// TwinCAT 3 PLC project TcLog
// Title: TcLog
// Company: Benedikt Geisler
// Author: Benedikt Geisler
// ProjectVersion: 0.6.1
// Description: TcLog provides logging functionality to TwinCAT.
// ProgramVersion: 3.1.4026.20
// libraries:
//   Tc2_Standard, * (Beckhoff Automation GmbH)
//   Tc2_System, * (Beckhoff Automation GmbH)
//   Tc2_Utilities, * (Beckhoff Automation GmbH)
//   Tc3_DynamicMemory, * (Beckhoff Automation GmbH)
//   Tc3_Module, * (Beckhoff Automation GmbH)
//   TcUnit, * (www.tcunit.org)
// project tree:
//   / Constants.TcGVL
//   Logger/ LogLevelToAdsLogMsgType.TcPOU (not stored), TcLog.TcPOU, TcLogCore.TcPOU (not stored), TcLogTrig.TcPOU (not stored)
//   StringBuilder/_Interfaces/ ILimitedStringBuilder.TcIO (not stored), IStringBuilder.TcIO (not stored)
//   Utils/ AnyToString.TcPOU (not stored), DateTime.TcPOU (not stored), DeleteOldFiles.TcPOU (not stored), DynamicStringBuffer.TcPOU (not stored), GetFileAgeInSeconds.TcPOU (not stored)
//   Utils/DataTypes/ DeleteFilesState.TcDUT (not stored), PersistToFileState.TcDUT (not stored)
//   Logger/DataTypes/ ErrorCodes.TcDUT (not stored), LogLevels.TcDUT (not stored), RollingIntervals.TcDUT (not stored), Error.TcDUT (not stored), LoggingConfiguration.TcDUT (not stored)
//   Logger/Interfaces/ ILog.TcIO (not stored), ILogCore.TcIO (not stored)
//   StringBuilder/ StringBuilder.TcPOU (not stored)
// real-time tasks:
//   TASK PlcTask1: cycle T#10ms, priority 21, ADS port 351

// ---- Constants.TcGVL
{attribute 'qualified_only'}
VAR_GLOBAL CONSTANT
	/// Fifo overhead needed to manage the string buffer
	FifoOverhead : UDINT := 10;

	/// Buffer size of temporary buffer used to persist all log messages in one cycle. 
	BufferSize : UDINT := (100 * (Tc2_System.MAX_STRING_LENGTH + FifoOverhead));
END_VAR

// ---- Logger/TcLog.TcPOU
/// `TcLog` is the client side of the logger.  
///
/// It is used to send the logs to `TcLogCore`. Typically, it is instantiated
/// once in each `FUNCTION_BLOCK` or `PROGRAM` where logging is done. The same 
/// instance can then be used for all logging within that POU. 
///
/// `TcLog` implements a string builder that facilitates the compilation of the log
/// message without the need for external data type conversions or multiple chained `CONCAT` calls.
/// See the method section for more information.
///
/// The last method to call after the log message has been built is one of ´[Debug|Information|Warning|Error|Fatal]`. 
/// This sets the log level of the message and sends it off to the log message queue of `TcLogCore` where it will
/// be processed according to its configuration.
{attribute 'linkalways'}
{attribute 'hide_all_locals'}
{attribute 'reflection'} 
FUNCTION_BLOCK TcLog IMPLEMENTS ILog
VAR
  _logConditionSatisfied : BOOL; // flag that indicates, whether log condition has been satisfied.
                                // Logging will only be carried out it this evaluates to TRUE.                    
  _logDataInitialized : BOOL; // flag that indicate, whether log data has been initialized.
                             // Necessary for configuration methods to provide a fluent interface.                            
  _logData : Tc2_System.T_MaxString; // contains message to be logged.
  _usedLogger : ILogCore;
  {attribute 'instance-path'} 
  {attribute 'noinit'} 
  _instancePath : STRING; // contains instance path
END_VAR
VAR_STAT
  {attribute 'hide'}
  s_loggerSingletonInstance : ILogCore; // Wires up TcLog ("Client") to TcLogCore ("Server") (Singleton-Behaviour)
END_VAR
VAR CONSTANT
  InvalidLoggerReference : UDINT := 0;
END_VAR

/// Appends any given data to the log string. The type of the provided data
/// has to be one of the [standard data types](https://infosys.beckhoff.com/english.php?content=../content/1033/tc3_plc_intro/2529388939.html&id=).
/// This method can be chained.
METHOD AppendAny : REFERENCE TO TcLog
VAR_INPUT
  /// data to be appended to log string.
  data : ANY;
END_VAR
InitializeLogData();

_logData := Tc2_Standard.CONCAT(_logData, AnyToString(data));

AppendAny REF= THIS^;
END_METHOD

/// Appends a BYTE to the log string.
/// This method can be chained.
METHOD PUBLIC AppendByte : REFERENCE TO TcLog
VAR_INPUT
  /// data to be appended to log string.
  data : BYTE;
END_VAR
AppendByte REF= AppendString(TO_STRING(data));
END_METHOD

/// Appends a DATE to the log string.
/// This method can be chained.
METHOD PUBLIC AppendDate : REFERENCE TO TcLog
VAR_INPUT
  /// data to be appended to log string.
  data : DATE;
END_VAR
AppendDate REF= AppendString(TO_STRING(data));
END_METHOD

/// Appends a DATE_AND_TIME to the log string.
/// This method can be chained.
METHOD PUBLIC AppendDateAndTime : REFERENCE TO TcLog
VAR_INPUT
  /// data to be appended to log string.
  data : DATE_AND_TIME;
END_VAR
AppendDateAndTime REF= AppendString(TO_STRING(data));
END_METHOD

/// Appends a DINT to the log string.
/// This method can be chained.
METHOD PUBLIC AppendDint : REFERENCE TO TcLog
VAR_INPUT
  /// data to be appended to log string.
  data : DINT;
END_VAR
AppendDint REF= AppendString(TO_STRING(data));
END_METHOD

/// Appends a DWORD to the log string.
/// This method can be chained.
METHOD PUBLIC AppendDword : REFERENCE TO TcLog
VAR_INPUT
  /// data to be appended to log string.
  data : DWORD;
END_VAR
AppendDword REF= AppendString(TO_STRING(data));
END_METHOD

/// Appends an INT to the log string.
/// This method can be chained.
METHOD PUBLIC AppendInt : REFERENCE TO TcLog
VAR_INPUT
  /// data to be appended to log string.
  data : INT;
END_VAR
AppendInt REF= AppendString(TO_STRING(data));
END_METHOD

/// Appends a LDATE to the log string.
/// This method can be chained.
METHOD PUBLIC AppendLDate : REFERENCE TO TcLog
VAR_INPUT
  /// data to be appended to log string.
  data : LDATE;
END_VAR
AppendLDate REF= AppendString(TO_STRING(data));
END_METHOD

/// Appends a LDATE_AND_TIME to the log string.
/// This method can be chained.
METHOD PUBLIC AppendLDateAndTime : REFERENCE TO TcLog
VAR_INPUT
  /// data to be appended to log string.
  data : LDATE_AND_TIME;
END_VAR
AppendLDateAndTime REF= AppendString(TO_STRING(data));
END_METHOD

/// Appends an LINT to the log string.
/// This method can be chained.
METHOD PUBLIC AppendLint : REFERENCE TO TcLog
VAR_INPUT
  /// data to be appended to log string.
  data : LINT;
END_VAR
AppendLint REF= AppendString(TO_STRING(data));
END_METHOD

/// Appends an LREAL to the log string.
/// This method can be chained.
METHOD PUBLIC AppendLreal : REFERENCE TO TcLog
VAR_INPUT
  /// data to be appended to log string.
  data : LREAL;
END_VAR
AppendLreal REF= AppendString(TO_STRING(data));
END_METHOD

/// Appends a LTIME_OF_DAY to the log string.
/// This method can be chained.
METHOD PUBLIC AppendLTimeOfDay : REFERENCE TO TcLog
VAR_INPUT
  /// data to be appended to log string.
  data : LTIME_OF_DAY;
END_VAR
AppendLTimeOfDay REF= AppendString(TO_STRING(data));
END_METHOD

/// Appends an LWORD to the log string.
/// This method can be chained.
METHOD PUBLIC AppendLword : REFERENCE TO TcLog
VAR_INPUT
  /// data to be appended to log string.
  data : LWORD;
END_VAR
AppendLword REF= AppendString(TO_STRING(data));
END_METHOD

/// Appends a REAL to the log string.
/// This method can be chained.
METHOD PUBLIC AppendReal : REFERENCE TO TcLog
VAR_INPUT
  /// data to be appended to log string.
  data : REAL;
END_VAR
AppendReal REF= AppendString(TO_STRING(data));
END_METHOD

/// Appends a SINT to the log string.
/// This method can be chained.
METHOD PUBLIC AppendSint : REFERENCE TO TcLog
VAR_INPUT
  /// data to be appended to log string.
  data : SINT;
END_VAR
AppendSint REF= AppendString(TO_STRING(data));
END_METHOD

/// Appends another string to the log message.
/// This method can be chained.
METHOD AppendString : REFERENCE TO TcLog
VAR_INPUT
  /// data to be appended to log string.
  data : Tc2_System.T_MaxString; 
END_VAR
InitializeLogData();

_logData := Tc2_Standard.CONCAT(_logData, data);
  
AppendString REF= THIS^;
END_METHOD

/// Appends a TIME_OF_DAY to the log string.
/// This method can be chained.
METHOD PUBLIC AppendTimeOfDay : REFERENCE TO TcLog
VAR_INPUT
  /// data to be appended to log string.
  data : TIME_OF_DAY;
END_VAR
AppendTimeOfDay REF= AppendString(TO_STRING(data));
END_METHOD

/// Appends a UDINT to the log string.
/// This method can be chained.
METHOD PUBLIC AppendUdint : REFERENCE TO TcLog
VAR_INPUT
  /// data to be appended to log string.
  data : UDINT;
END_VAR
AppendUdint REF= AppendString(TO_STRING(data));
END_METHOD

/// Appends a UINT to the log string.
/// This method can be chained.
METHOD PUBLIC AppendUint : REFERENCE TO TcLog
VAR_INPUT
  /// data to be appended to log string.
  data : UINT;
END_VAR
AppendUint REF= AppendString(TO_STRING(data));
END_METHOD

/// Appends a ULINT to the log string.
/// This method can be chained.
METHOD PUBLIC AppendUlint : REFERENCE TO TcLog
VAR_INPUT
  /// data to be appended to log string.
  data : ULINT;
END_VAR
AppendUlint REF= AppendString(TO_STRING(data));
END_METHOD

/// Appends a USINT to the log string.
/// This method can be chained.
METHOD PUBLIC AppendUsint : REFERENCE TO TcLog
VAR_INPUT
  /// data to be appended to log string.
  data : USINT;
END_VAR
AppendUsint REF= AppendString(TO_STRING(data));
END_METHOD

/// Appends information about the given variable to the log string. 
/// This method can be chained.
/// Example: 

/// ```st
/// VAR
///   Logger: TcLog;
///    myInt : INT := 10;
///   myVarInfo : __SYSTEM.VAR_INFO := __VARINFO(myInt);
/// END_VAR
/// Logger.AppendVariable(myVarInfo, myInt);
/// ```
///
METHOD AppendVariable : REFERENCE TO TcLog
VAR_INPUT
  /// [VAR_INFO](https://infosys.beckhoff.com/index.php?content=../content/1031/tc3_plc_intro/3527777675.html&id=) of variable to be appended to log string.
  varInfo : __SYSTEM.VAR_INFO;
  /// Value of variable to be appended to log string.
  value : ANY; 
END_VAR
VAR
  format : Tc2_Utilities.FB_FormatString;
  symbolName : Tc2_System.T_MaxString;
  typeName : Tc2_System.T_MaxString;
END_VAR
InitializeLogData();

symbolName := varInfo.Symbol;
typeName := varInfo.TypeName; 

format(
  sFormat := '%s [%s] : ',
  arg1 := Tc2_Utilities.F_String(symbolName),
  arg2 := Tc2_Utilities.F_String(typeName));
  
AppendString(format.sOut);
AppendAny(value);

AppendVariable REF= THIS^;
END_METHOD

/// Appends a WORD to the log string.
/// This method can be chained.
METHOD PUBLIC AppendWord : REFERENCE TO TcLog
VAR_INPUT
  /// data to be appended to log string.
  data : WORD;
END_VAR
AppendWord REF= AppendString(TO_STRING(data));
END_METHOD

/// Logs the log string in DEBUG level.
METHOD Debug : BOOL
VAR_INPUT
  /// Message to be appended to log string.
  message : Tc2_System.T_MaxString; 
END_VAR
InitializeLogData();
IF _logConditionSatisfied THEN
  IF _usedLogger <> InvalidLoggerReference THEN 
    _usedLogger.LogStandardFormat(Tc2_Standard.CONCAT(_logData, message), ShortenInstancePath(_instancePath), LogLevels.Debug); 
  ELSE
    Tc2_System.ADSLOGSTR(ADSLOG_MSGTYPE_LOG OR LogLevelToAdsLogMsgType(LogLevels.Error), 'usedLogger: No valid reference', ''); 
  END_IF
END_IF
_logDataInitialized := FALSE;
END_METHOD

/// Logs the log string in ERROR level.
METHOD Error : BOOL
VAR_INPUT
  /// Message to be appended to log string.
  message : Tc2_System.T_MaxString; 
END_VAR
InitializeLogData();
IF _logConditionSatisfied THEN
  IF _usedLogger <> InvalidLoggerReference THEN 
    _usedLogger.LogStandardFormat(Tc2_Standard.CONCAT(_logData, message), ShortenInstancePath(_instancePath), LogLevels.Error); 
  ELSE
    Tc2_System.ADSLOGSTR(ADSLOG_MSGTYPE_LOG OR LogLevelToAdsLogMsgType(LogLevels.Error), 'usedLogger: No valid reference', ''); 
  END_IF
END_IF
_logDataInitialized := FALSE;
END_METHOD

/// Logs the log string in FATAL level.
METHOD Fatal : BOOL
VAR_INPUT
  /// Message to be appended to log string.
  message : Tc2_System.T_MaxString; 
END_VAR
InitializeLogData();
IF _logConditionSatisfied THEN
  IF _usedLogger <> InvalidLoggerReference THEN 
    _usedLogger.LogStandardFormat(Tc2_Standard.CONCAT(_logData, message), ShortenInstancePath(_instancePath), LogLevels.Fatal); 
  ELSE
    Tc2_System.ADSLOGSTR(ADSLOG_MSGTYPE_LOG OR LogLevelToAdsLogMsgType(LogLevels.Error), 'usedLogger: No valid reference', ''); 
  END_IF
END_IF
_logDataInitialized := FALSE;
END_METHOD

/// Logs the log string in INFORMATION level.
METHOD Information : BOOL
VAR_INPUT
  /// Message to be appended to log string.
  message : Tc2_System.T_MaxString; 
END_VAR
InitializeLogData();
IF _logConditionSatisfied THEN
  IF _usedLogger <> InvalidLoggerReference THEN 
    _usedLogger.LogStandardFormat(Tc2_Standard.CONCAT(_logData, message), ShortenInstancePath(_instancePath), LogLevels.Information); 
  ELSE
    Tc2_System.ADSLOGSTR(ADSLOG_MSGTYPE_LOG OR LogLevelToAdsLogMsgType(LogLevels.Error), 'usedLogger: No valid reference', ''); 
  END_IF
END_IF
_logDataInitialized := FALSE;
END_METHOD

/// Initializes the reference to the core logger. Should only be called once from the core logger directly.
METHOD PUBLIC Init : BOOL
VAR_INPUT
  /// Reference to TcLoggerCore instance.
  ref2Core : ILogCore; 
END_VAR
IF s_loggerSingletonInstance = 0 THEN
	s_loggerSingletonInstance := ref2Core;
END_IF
END_METHOD

// Necessary to provide a fluent interface of the function. 
// Has to be called at the begin of any method that returns a reference to THIS^
METHOD PRIVATE InitializeLogData : BOOL
IF NOT _logDataInitialized THEN
  _logConditionSatisfied := TRUE;
  _logData := '';
  _logDataInitialized := TRUE;
  IF _usedLogger = 0 THEN _usedLogger := s_loggerSingletonInstance; END_IF
END_IF
END_METHOD

/// Conditional execution of the log command. Only executes logging when Cond = TRUE.
METHOD OnCondition : REFERENCE TO TcLog
VAR_INPUT
  /// Logs data only if this condition evaluates to TRUE.
  cond : BOOL; 
END_VAR
InitializeLogData();

_logConditionSatisfied := cond;

OnCondition REF= THIS^;
END_METHOD

/// Initializes the reference to the core logger. This enables you to use several
/// loggers with different configurations in one project.
METHOD SetLogger : BOOL
VAR_INPUT
  /// Reference to Core Logger
  ref2Core : ILogCore; 
END_VAR
_usedLogger := ref2Core;
END_METHOD

// Helper method. Shortens the instance path by omitting superfluent information
// such as concrete logger instance and plc/project names.
{attribute 'hide'}
METHOD PRIVATE ShortenInstancePath : Tc2_System.T_MaxString
VAR_INPUT
  path : Tc2_System.T_MaxString; // Instance path to be shortened.
END_VAR
VAR
  i : UINT;
  shortenedPath : Tc2_System.T_MaxString;
  positionInString : INT := 0;
  positionOfLastDot : INT := 0;
END_VAR
shortenedPath := path;

// Find last '.'
WHILE(Tc2_Standard.FIND(shortenedPath, '.') > 0) DO
  positionInString := Tc2_Standard.FIND(shortenedPath, '.');
  shortenedPath := Tc2_Standard.DELETE(shortenedPath, positionInString+1, 0); 
  positionOfLastDot := positionOfLastDot+positionInString;
END_WHILE

shortenedPath := Path;
// Delete instantiation of this FB (obvious information)
shortenedPath := Tc2_Standard.DELETE(shortenedPath, Tc2_Standard.LEN(shortenedPath)-positionOfLastDot+1, positionOfLastDot);
// Delete project information
positionInString := Tc2_Standard.FIND(shortenedPath, '.');
shortenedPath := Tc2_Standard.DELETE(shortenedPath, positionInString+1, 0);
// Delete PLC information
positionInString := Tc2_Standard.FIND(shortenedPath, '.');
shortenedPath := Tc2_Standard.DELETE(shortenedPath, positionInString+1, 0);

ShortenInstancePath := shortenedPath;
END_METHOD

/// Logs directly to ADS log, ignoring the settings of the base logger.
METHOD ToAdsLog : BOOL
VAR_INPUT
  /// Log level in which message should be logged to ADS.
  logLevel : LogLevels; 
END_VAR
InitializeLogData();

IF _logConditionSatisfied THEN
  Tc2_System.ADSLOGSTR(ADSLOG_MSGTYPE_LOG OR LogLevelToAdsLogMsgType(logLevel), _logData, ''); 
END_IF

_logDataInitialized := FALSE;
END_METHOD

/// Saves custom formatted log string. 
/// No addtitional information will be added, no formatting will be applied.
METHOD ToCustomFormat : BOOL
VAR_INPUT
  /// Message to be appended to log string.
  message : Tc2_System.T_MaxString; 
END_VAR
InitializeLogData();
IF _logConditionSatisfied THEN
  IF _usedLogger <> InvalidLoggerReference THEN 
    _usedLogger.LogCustomFormat(Tc2_Standard.CONCAT(_logData, message)); 
  ELSE
    Tc2_System.ADSLOGSTR(ADSLOG_MSGTYPE_LOG OR LogLevelToAdsLogMsgType(LogLevels.Error), 'usedLogger: No valid reference', ''); 
  END_IF
END_IF
_logDataInitialized := FALSE;
END_METHOD

/// Logs the log string in WARNING level.
METHOD Warning : BOOL
VAR_INPUT
  /// Message to be appended to log string.
  message : Tc2_System.T_MaxString; 
END_VAR
InitializeLogData();
IF _logConditionSatisfied THEN
  IF _usedLogger <> InvalidLoggerReference THEN 
    _usedLogger.LogStandardFormat(Tc2_Standard.CONCAT(_logData, message), ShortenInstancePath(_instancePath), LogLevels.Warning); 
  ELSE
    Tc2_System.ADSLOGSTR(ADSLOG_MSGTYPE_LOG OR LogLevelToAdsLogMsgType(LogLevels.Error), 'usedLogger: No valid reference', ''); 
  END_IF
END_IF
_logDataInitialized := FALSE;
END_METHOD

END_FUNCTION_BLOCK
